FUNCTION InvertFactor : LREAL
VAR_INPUT
	EN: BOOL;
	Val: LREAL;
END_VAR
VAR
END_VAR

IF EN THEN
	InvertFactor := LIMIT(0, 1 - LIMIT(0, Val, 1), 1);
ELSE
	InvertFactor := Val;
END_IF

END_FUNCTION

(* stored: Version 1.1.0.1, ProductVersion 3.1.4024.6
   POU InvertFactor: Id {e9cc6063-8859-476f-bc2e-ee3dc412804a}, SpecialFunc None *)
